PROGRAM LADDER1
VAR
	stop: BOOL;
	start: BOOL;
	emergency: BOOL;
	S_place: BOOL;
	S_full: BOOL;
	S_empty: BOOL;
	S_loading: BOOL;
	S_unload: BOOL;
	valve: BOOL;
	Motor: BOOL;
	y1: BOOL;
	y3: BOOL;
	y2:BOOL;
	TankEmpty: BOOL;
    CU: BOOL; 
    RESET: BOOL; 
    PV: WORD; 
	FILLING: BOOL;
	CV: WORD;
	Q: Bool;
	counter: CTU;
END_VAR
VAR // added by the converter: edge detectors and wires of the graphical bodies
    _w1, _w2 : BOOL;
END_VAR

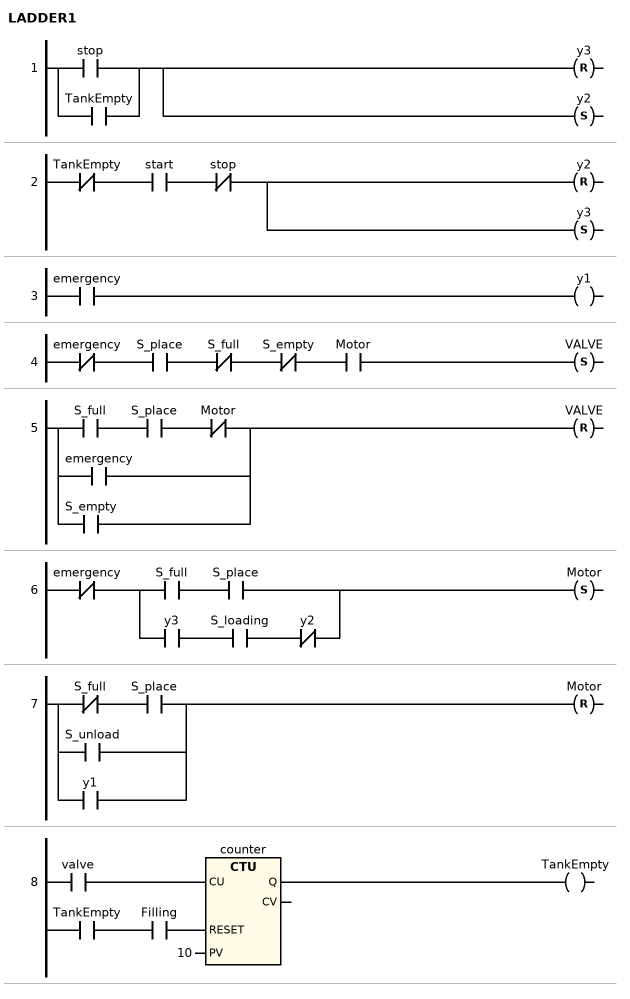
// NETWORK 1
_w1 := stop OR TankEmpty;
y3 R= _w1;
y2 S= _w1;

// NETWORK 2
_w2 := NOT TankEmpty AND start AND NOT stop;
y2 R= _w2;
y3 S= _w2;

// NETWORK 3
y1 := emergency;

// NETWORK 4
VALVE S= NOT emergency AND S_place AND NOT S_full AND NOT S_empty AND Motor;

// NETWORK 5
VALVE R= S_full AND S_place AND NOT Motor OR emergency OR S_empty;

// NETWORK 6
Motor S= NOT emergency AND (S_full AND S_place OR y3 AND S_loading AND NOT y2);

// NETWORK 7
Motor R= NOT S_full AND S_place OR S_unload OR y1;

// NETWORK 8
counter(CU := valve, RESET := TankEmpty AND Filling, PV := 10); // CTU
TankEmpty := counter.Q;

END_PROGRAM

(* stored: Version 1.1.0.1, ProductVersion 3.1.4020.6
   POU LADDER1: Id {b96b3cff-5724-4696-ad41-d629b3720a9f}, SpecialFunc None *)
